INTERFACE I_Simulatable EXTENDS I_Base

{attribute 'monitoring' := 'call'}
PROPERTY Simulated : BOOL
GET
END_GET
SET
END_SET
END_PROPERTY

END_INTERFACE

(* stored: Version 1.1.0.1, ProductVersion 3.1.4026.18
   Itf I_Simulatable: Id {b2009768-caaa-4ccc-a400-96e337139a16}
   Property Simulated: Id {09d92c05-d7d0-4ed4-add0-3613eebc0c68}
   Get Get: Id {86255679-f41c-44e9-b682-4b6322219af1}
   Set Set: Id {ee1753cd-c3b1-4015-9708-8c4040af9ca4} *)
